{attribute 'GeneratedUsingTerminal: EL5002-0000-0016'}
{attribute addProperty BoxType "EL5002-0000-0016"}
{attribute addProperty Id "StatusAT %I*Status_ACC8459F6Counter_valueAT %I*UDINT4"}
{attribute addProperty CRC "238915123"}
{attribute addProperty Size "10"}
TYPE SSI_Inputs_Channel_0E3D8E33 :
STRUCT
	{attribute addProperty Name "Status"}
	Status AT %I* : Status_ACC8459F;
	{attribute addProperty Name "Counter_value"}
	Counter_value AT %I* : UDINT;
END_STRUCT
END_TYPE

(* stored: Version 1.2.0.0, ProductVersion 3.1.4024.9
   DUT SSI_Inputs_Channel_0E3D8E33: Id {c71f908f-ff0a-493e-b31a-919283503a32} *)
